_CFC_ (* Continuous Function Chart, elements in execution order *)
#0 AND(NOT SCHU_P2_2_TS1_DI5, SCHU_P2_2_KV1_DI4)
#1 TON_Kv1_1:TON(IN: #0, PT: T#10s)
#2 RT_PUSK_OLD:R_TRIG(CLK: #1.Q)
#3 AND(#2.Q, OLD_SOST)
#4 AND(NOT SCHU_P2_2_TE2_M_ZASCH, SCHU_P2_2_KV1_DI4)
#5 TON_Kv1_11:TON(IN: #4, PT: T#10s)
#6 RT_PUSK_OLD1:R_TRIG(CLK: #5.Q)
#7 AND(#6.Q, OLD_SOST)
#8 OR(SCHU_P2_2_UST_PUSK_VH, #3, #7)
#9 AND(NOT SCHU_P2_2_UST_RE_OSTANOV, #8)
#10 RT_STOP:R_TRIG(CLK: SCHU_P2_2_UST_STOP_VH)
#11 OR(#10.Q, SCHU_P2_2_UST_SET_STOP, SCHU_P2_2_UST_SET_OSTANOV)
#12 RS_Sost:RS(SET: #9, RESET1: #11)
#13 SCHU_P2_2_UST_SOST_VKL <= #12.Q1
#14 SCHU_P2_2_UST_SOST_OTKL <= NOT #12.Q1
#15 AND(NOT SCHU_P2_2_TS1_DI5, SCHU_P2_2_KV1_DI4)
#16 TON_Kv11:TON(IN: #15, PT: T#1.5m)
#17 AND(NOT SCHU_P2_2_TE2_M_ZASCH, SCHU_P2_2_KV1_DI4)
#18 TON_Kv1:TON(IN: #17, PT: T#1.5m)
#19 AND(#16.Q, #18.Q)
#20 AND(#12.Q1, #19)
#21 AND(NOT #12.Q1, #19)
#22 CTU_TS:CTU(CU: SCHU_P2_2_TS1_DI5, RESET: #22.Q, PV: 3)
#23 =(#22.CV, 0)
#24 AND(#23, SCHU_P2_2_TS1_DI5)
#25 TOF_TS_1:TOF(IN: #24, PT: T#60m)
#26 =(#22.CV, 1)
#27 AND(#26, SCHU_P2_2_TS1_DI5)
#28 TOF_TS_2:TOF(IN: #27, PT: T#60m)
#29 =(#22.CV, 2)
#30 AND(#29, SCHU_P2_2_TS1_DI5)
#31 TOF_TS_3:TOF(IN: #30, PT: T#60m)
#32 AND(#25.Q, #28.Q, #31.Q)
#33 CTU_Te:CTU(CU: SCHU_P2_2_TE2_M_ZASCH, RESET: #33.Q, PV: 3)
#34 =(#33.CV, 0)
#35 AND(#34, SCHU_P2_2_TE2_M_ZASCH)
#36 TOF_TE_1:TOF(IN: #35, PT: T#60m)
#37 =(#33.CV, 1)
#38 AND(#37, SCHU_P2_2_TE2_M_ZASCH)
#39 TOF_Te_2:TOF(IN: #38, PT: T#60m)
#40 =(#33.CV, 2)
#41 AND(#40, SCHU_P2_2_TE2_M_ZASCH)
#42 TOF_Te_3:TOF(IN: #41, PT: T#60m)
#43 AND(#36.Q, #39.Q, #42.Q)
#44 OR(#21, #32, #43)
#45 RS_Old_Sost:RS(SET: #20, RESET1: #44)
#46 OLD_SOST <= #45.Q1
_END_CFC_
END_PROGRAM

(* POU Regim/Stop, CFC *)
PROGRAM Stop
VAR
	FT_Ostanov: F_TRIG;
	sr_stop: SR;
	TOF_Progrev: TOF;
END_VAR
VAR (* helpers for the ST form of the networks *)
	_t19 : BOOL;
END_VAR
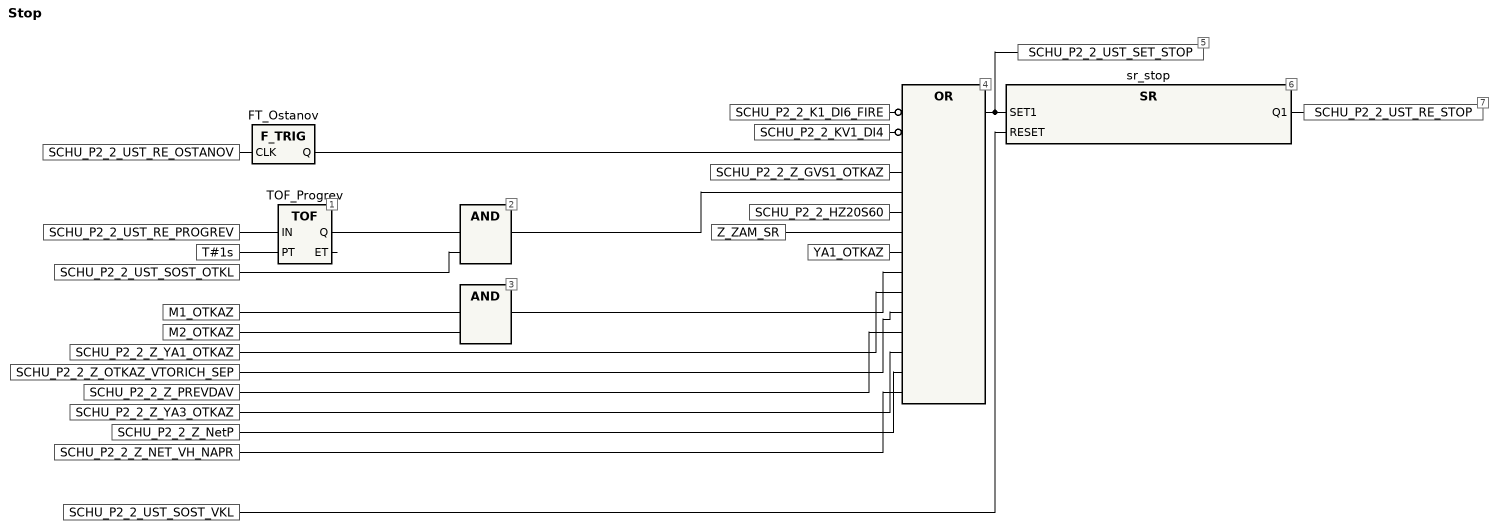
_CFC_ (* Continuous Function Chart, elements in execution order *)
#0 FT_Ostanov:F_TRIG(CLK: SCHU_P2_2_UST_RE_OSTANOV)
#1 TOF_Progrev:TOF(IN: SCHU_P2_2_UST_RE_PROGREV, PT: T#1s)
#2 AND(#1.Q, SCHU_P2_2_UST_SOST_OTKL)
#3 AND(M1_OTKAZ, M2_OTKAZ)
#4 OR(NOT SCHU_P2_2_K1_DI6_FIRE, NOT SCHU_P2_2_KV1_DI4, #0.Q, SCHU_P2_2_Z_GVS1_OTKAZ, #2, SCHU_P2_2_HZ20S60, Z_ZAM_SR, YA1_OTKAZ, #3, SCHU_P2_2_Z_YA1_OTKAZ, SCHU_P2_2_Z_OTKAZ_VTORICH_SEP, SCHU_P2_2_Z_PREVDAV, SCHU_P2_2_Z_YA3_OTKAZ, SCHU_P2_2_Z_NetP, SCHU_P2_2_Z_NET_VH_NAPR)
#5 SCHU_P2_2_UST_SET_STOP <= #4
#6 sr_stop:SR(SET1: #4, RESET: SCHU_P2_2_UST_SOST_VKL)
#7 SCHU_P2_2_UST_RE_STOP <= #6.Q1
_END_CFC_
(* the same logic as Structured Text *)
FT_Ostanov(CLK := SCHU_P2_2_UST_RE_OSTANOV);
TOF_Progrev(IN := SCHU_P2_2_UST_RE_PROGREV, PT := T#1s);
_t19 := NOT SCHU_P2_2_K1_DI6_FIRE OR NOT SCHU_P2_2_KV1_DI4 OR FT_Ostanov.Q OR SCHU_P2_2_Z_GVS1_OTKAZ OR (TOF_Progrev.Q AND SCHU_P2_2_UST_SOST_OTKL) OR SCHU_P2_2_HZ20S60 OR Z_ZAM_SR OR YA1_OTKAZ OR (M1_OTKAZ AND M2_OTKAZ) OR SCHU_P2_2_Z_YA1_OTKAZ OR SCHU_P2_2_Z_OTKAZ_VTORICH_SEP OR SCHU_P2_2_Z_PREVDAV OR SCHU_P2_2_Z_YA3_OTKAZ OR SCHU_P2_2_Z_NetP OR SCHU_P2_2_Z_NET_VH_NAPR;
SCHU_P2_2_UST_SET_STOP := _t19;
sr_stop(SET1 := _t19, RESET := SCHU_P2_2_UST_SOST_VKL);
SCHU_P2_2_UST_RE_STOP := sr_stop.Q1;
END_PROGRAM

(* POU Regim/Ostanov, CFC *)
PROGRAM Ostanov
VAR
	RT_OTKL: R_TRIG;
	SR_OSTANOV: SR;
	TON_AVR_M: TON;
	Z_zam_ostatov: R_TRIG;
END_VAR
VAR (* helpers for the ST form of the networks *)
	_t31 : BOOL;
END_VAR
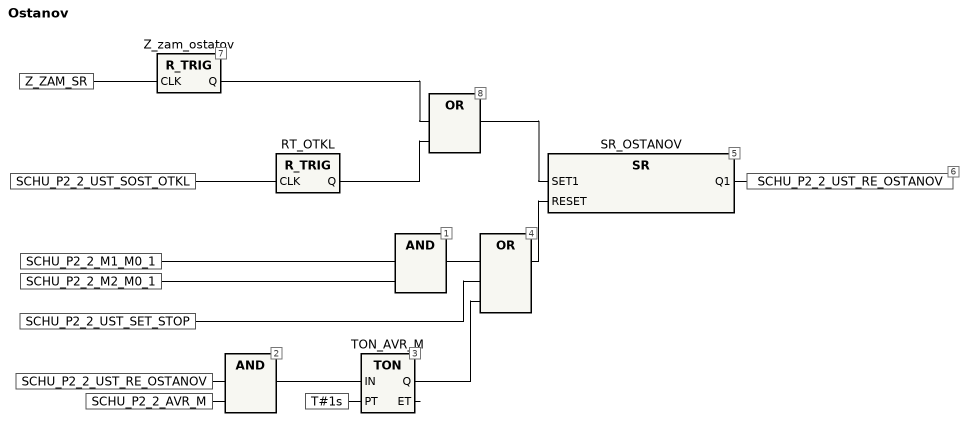
_CFC_ (* Continuous Function Chart, elements in execution order *)
#0 RT_OTKL:R_TRIG(CLK: SCHU_P2_2_UST_SOST_OTKL)
#1 AND(SCHU_P2_2_M1_M0_1, SCHU_P2_2_M2_M0_1)
#2 AND(SCHU_P2_2_UST_RE_OSTANOV, SCHU_P2_2_AVR_M)
#3 TON_AVR_M:TON(IN: #2, PT: T#1s)
#4 OR(#1, SCHU_P2_2_UST_SET_STOP, #3.Q)
#5 SR_OSTANOV:SR(SET1: #8, RESET: #4)
#6 SCHU_P2_2_UST_RE_OSTANOV <= #5.Q1
#7 Z_zam_ostatov:R_TRIG(CLK: Z_ZAM_SR)
#8 OR(#7.Q, #0.Q)
_END_CFC_
(* the same logic as Structured Text *)
RT_OTKL(CLK := SCHU_P2_2_UST_SOST_OTKL);
TON_AVR_M(IN := SCHU_P2_2_UST_RE_OSTANOV AND SCHU_P2_2_AVR_M, PT := T#1s);
SR_OSTANOV(SET1 := _t31, RESET := (SCHU_P2_2_M1_M0_1 AND SCHU_P2_2_M2_M0_1) OR SCHU_P2_2_UST_SET_STOP OR TON_AVR_M.Q);
SCHU_P2_2_UST_RE_OSTANOV := SR_OSTANOV.Q1;
Z_zam_ostatov(CLK := Z_ZAM_SR);
_t31 := Z_zam_ostatov.Q OR RT_OTKL.Q;
END_PROGRAM

(* POU Regim/Progrev, CFC *)
PROGRAM Progrev
VAR
	RS_Progrev: RS;
	RT_VKL: R_TRIG;
	TON_SCHU_P2_2_TE2_M_UST: TON;
	SR_First_On: SR;
END_VAR
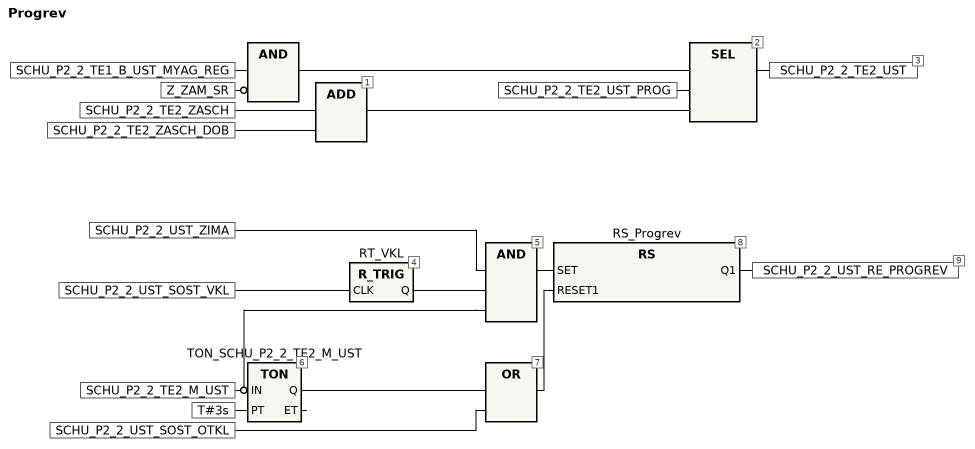
_CFC_ (* Continuous Function Chart, elements in execution order *)
#0 AND(SCHU_P2_2_TE1_B_UST_MYAG_REG, NOT Z_ZAM_SR)
#1 ADD(SCHU_P2_2_TE2_ZASCH, SCHU_P2_2_TE2_ZASCH_DOB)
#2 SEL(#0, SCHU_P2_2_TE2_UST_PROG, #1)
#3 SCHU_P2_2_TE2_UST <= #2
#4 RT_VKL:R_TRIG(CLK: SCHU_P2_2_UST_SOST_VKL)
#5 AND(SCHU_P2_2_UST_ZIMA, #4.Q, SCHU_P2_2_TE2_M_UST)
#6 TON_SCHU_P2_2_TE2_M_UST:TON(IN: NOT SCHU_P2_2_TE2_M_UST, PT: T#3s)
#7 OR(#6.Q, SCHU_P2_2_UST_SOST_OTKL)
#8 RS_Progrev:RS(SET: #5, RESET1: #7)
#9 SCHU_P2_2_UST_RE_PROGREV <= #8.Q1
_END_CFC_
(* the same logic as Structured Text *)
SCHU_P2_2_TE2_UST := SEL(SCHU_P2_2_TE1_B_UST_MYAG_REG AND NOT Z_ZAM_SR, SCHU_P2_2_TE2_UST_PROG, SCHU_P2_2_TE2_ZASCH + SCHU_P2_2_TE2_ZASCH_DOB);
RT_VKL(CLK := SCHU_P2_2_UST_SOST_VKL);
TON_SCHU_P2_2_TE2_M_UST(IN := NOT SCHU_P2_2_TE2_M_UST, PT := T#3s);
RS_Progrev(SET := SCHU_P2_2_UST_ZIMA AND RT_VKL.Q AND SCHU_P2_2_TE2_M_UST, RESET1 := TON_SCHU_P2_2_TE2_M_UST.Q OR SCHU_P2_2_UST_SOST_OTKL);
SCHU_P2_2_UST_RE_PROGREV := RS_Progrev.Q1;
END_PROGRAM

(* POU Regim/Pusk, CFC *)
PROGRAM Pusk
VAR
	RS_Pusk: RS;
	FT_PROGREV: F_TRIG;
	RT_VKL: R_TRIG;
	TON_sost_VKL: TON;
	TON_AVR_M: TON;
	re_start: F_TRIG;
	TON_Z_ZAM: TON;
END_VAR
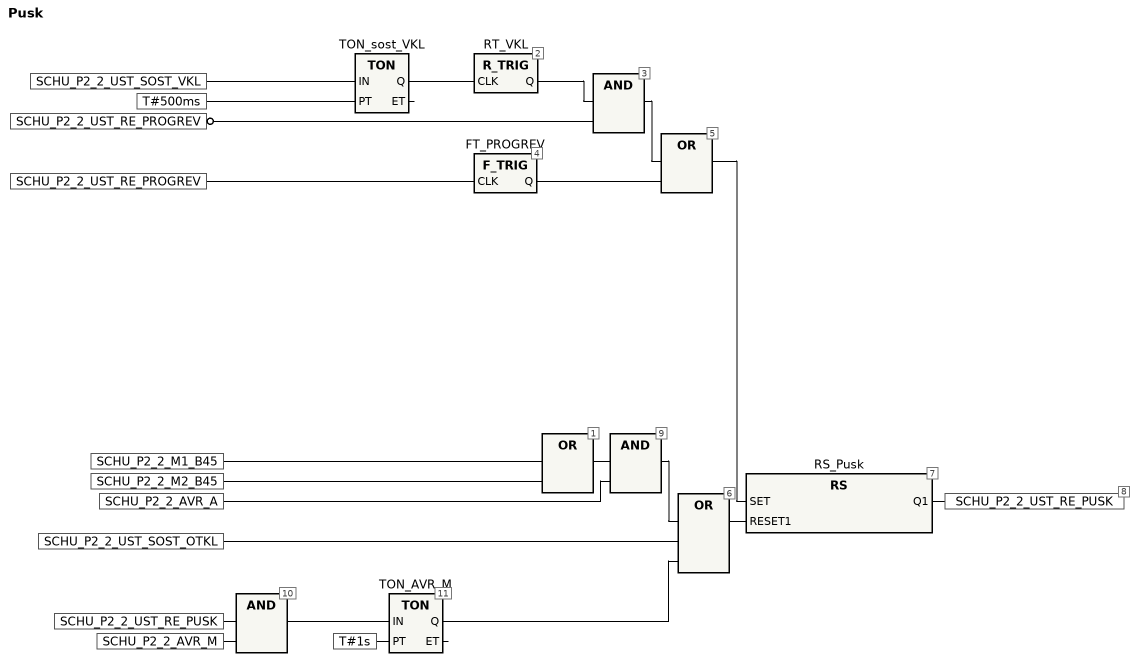
